FUNCTION_BLOCK Calibracao_V03
VAR_INPUT
	Flowmeter:REAL;
END_VAR
VAR_OUTPUT
	TurnOnPump:BOOL;
	Valv1:BOOL;
	Valv2:BOOL;
	Valv3:BOOL;
	Valv4:BOOL;
	PumpSpeed:REAL;	//Velocidade enviada para a bomba
END_VAR
VAR
	SwitchCase:INT;
	Start: BOOL;
	Stop: BOOL;
	TON_Temporizador1: TON;
	TON_Temporizador2: TON;
	BaixaVazao	:ARRAY[1..10] OF REAL;
	AltaVazao	:ARRAY[1..10] OF REAL;
	MediaBaixaVazao :REAL;
	MediaAltaVazao	:REAL;
	Counter: INT;
	i: INT;
	CoefAngular: REAL;
END_VAR

//Esse programa encontrará dois pontos relacionando vazão e velocidade (x e y), assim, será possível definir a função da bomba

IF Start AND NOT Stop  AND Seguridad.PB_Emergencia THEN
	SwitchCase := 10;
	Start := FALSE;
END_IF

IF STOP OR NOT Seguridad.PB_Emergencia THEN
	SwitchCase := 0;
	STOP := FALSE;
END_IF

//Temporizadores
TON_Temporizador1(PT:=T#5S);
TON_Temporizador2( IN:=TON_Temporizador1.Q AND NOT TON_Temporizador2.Q, PT:=T#1S);


CASE SwitchCase OF
	0:	//Desliga o sistema
		TurnOnPump := FALSE;
		Valv1 := FALSE;
		Valv2 := FALSE;
		Valv3 := FALSE;
		Valv4 := FALSE;
		
	10:	//Inicia a bomba com 20%
		PumpSpeed := 20;
		TurnOnPump := TRUE;
		TON_Temporizador1.IN := TRUE;
		
		//Após 5s da bomba ligada, a vazão é computada a cada 1s
		IF TON_Temporizador1.Q THEN
			Counter := 1;
			SwitchCase := 20;
		END_IF
		
	20:	//Cômputo da vazão com 10% da velocidade e aguarda a estabilização
		IF TON_Temporizador2.Q THEN
			IF Flowmeter > 0 THEN
				BaixaVazao[Counter] := Flowmeter;
				Counter := Counter + 1;
			END_IF
		END_IF
		IF Counter > 10 THEN
			TON_Temporizador1.IN := FALSE;
			SwitchCase := 30;
		END_IF
	
	30:	//Inicia a bomba com 80% e aguarda a estabilização
		PumpSpeed := 80;
		TON_Temporizador1.IN := TRUE;
		IF TON_Temporizador1.Q THEN
			Counter := 1;
			SwitchCase := 40;
		END_IF
		
	40:	//Cômputo da vazão com 80% da velocidade
		IF TON_Temporizador2.Q THEN
			IF Flowmeter > 0 THEN
				AltaVazao[Counter] := Flowmeter;
				Counter := Counter + 1;
			END_IF
		END_IF
		IF Counter > 10 THEN
			TON_Temporizador1.IN := FALSE;
			SwitchCase := 50;
		END_IF
		
	50:	//Cálculo das médias
		MediaBaixaVazao	:= 0;
		MediaAltaVazao	:= 0;
		FOR i := 1 TO 10 BY 1 DO
			MediaBaixaVazao	:= MediaBaixaVazao + BaixaVazao[i];
			MediaAltaVazao	:= MediaAltaVazao + AltaVazao[i];
		END_FOR
		MediaBaixaVazao	:= MediaBaixaVazao/10;
		MediaAltaVazao	:= MediaAltaVazao/10;
		
		//Cálculo do coeficiente angular
		CoefAngular := (MediaAltaVazao - MediaBaixaVazao)/(80 - 20);
		TurnOnPump := FALSE;
		SwitchCase := 0;
		
	60:	//
		
END_CASE

END_FUNCTION_BLOCK

(* stored: Version 1.1.0.1, ProductVersion 3.1.4024.14
   POU Calibracao_V03: Id {9c102509-397a-4bb3-aac4-4d63d182f1e4}, SpecialFunc None *)
